(* LS Electric XG5000 project: IEC300S *)
(* PLC LSPLC *)

PROGRAM NewProgram (* task: 스캔 프로그램 *)

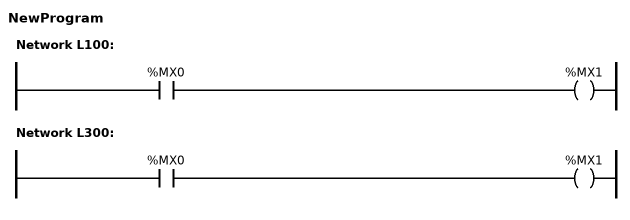
(* Rung L100 *)
%MX1 := %MX0;
(* Rung L300 *)
%MX1 := %MX0;
END_PROGRAM